(* PLC project CoDeSys External Library Template, WAGO e!COCKPIT e!COCKPIT, author 3S - Smart Software Solutions GmbH *)
(* stored: creationDateTime 2019-10-29T12:37:19.7827896, version 3.5.5.30, modificationDateTime 2019-10-29T12:36:39.3744516, organization 3S - Smart Software Solutions GmbH *)
(* Library project template with all possible element types, docu and a sample project structure *)

FUNCTION fnCRC16Wysylanie : WORD
  VAR_INPUT
    sKomunikat : alSTRINGKomunikat;
  END_VAR
  VAR_IN_OUT
    arTransmitterBuffer : ARRAY[1..512] OF BYTE;
    udiTransmitterNBytes : UDINT;
  END_VAR
  VAR
    intPetla : INT;
    wCRC16_modbus : WORD;
  END_VAR

            FOR intPetla := 1 TO LEN(sKomunikat) BY 1 DO
	arTransmitterBuffer[intPetla] := string_to_ASCIIByte(MID(sKomunikat , 1 , intPetla));
END_FOR

wCRC16_modbus := fnCRC16Obliczanie(sKomunikat);

arTransmitterBuffer[LEN(sKomunikat) + 1] := MEM.LowByte(wCRC16_modbus);
arTransmitterBuffer[LEN(sKomunikat) + 2] := MEM.HighByte(wCRC16_modbus);

udiTransmitterNBytes := INT_TO_UDINT(LEN(sKomunikat)) + 2;	

fnCRC16Wysylanie := wCRC16_modbus;
          
END_FUNCTION
